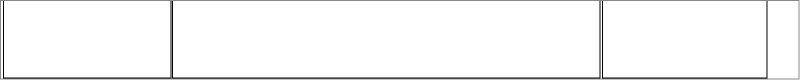
VISUALIZATION Header  // 800x80
    Rectangle (3,0 168x78)
    Rectangle (172,0 428x78)
    Rectangle (602,0 165x78)
END_VISUALIZATION

(* stored: Version 1.1.0.1, ProductVersion 3.1.4024.12
   Visu Header: Id {275838cf-745a-4e60-9f66-0ec34ac77d85} *)
